{attribute 'GeneratedUsingTerminal: AT2050-0500-0016'}
{attribute addProperty BoxType "AT2050-0500-0016"}
{attribute addProperty Id "A_0097_AT2025_5250_0018_AT2025_5250AT2025_01D6DEDF80"}
{attribute addProperty CRC "2164314109"}
{attribute addProperty Size "80"}
TYPE A_0047_AT2050_0500_0016_8100CFFD EXTENDS AT2050_86175B41 :
STRUCT
	{attribute addProperty Name "A_0097_AT2025_5250_0018_AT2025_5250"}
	{attribute addProperty PreviousPort "A_0047(AT2050-0500-0016) : B"}
	A_0097_AT2025_5250_0018_AT2025_5250 : AT2025_01D6DEDF;
END_STRUCT
END_TYPE

(* stored: Version 1.2.0.0, ProductVersion 3.1.4024.9
   DUT A_0047_AT2050_0500_0016_8100CFFD: Id {85ebff22-731f-4cbe-8bd1-edabdf551a09} *)
